(* IEC 61131-3 sources: ae-tiax/test/ParkingCounter, 2 files *)

(* ---- TestCounter.st ---- *)
USING Siemens.Ax.ExampleLibrary;
USING AxUnit;

NAMESPACE Siemens.Ax

    {TestFixture}
    CLASS TestCounter
        VAR
            c : Counter;
            cStateless : Counter;
        END_VAR

        // This method will be called before each test method
        {TestSetup}
        METHOD PUBLIC MyTestSetup
            c := cStateless;
        END_METHOD
        {Test}
        METHOD PUBLIC Test_CountUp_1_Time_And_Get_1
            c.CountUp();
            Assert.Equal(actual := c.GetValue(), expected := 1);
        END_METHOD
        {Test}
        METHOD PUBLIC Test_CountDown_1_Time_And_Get_Minus_1
            c.CountDown();
            Assert.Equal(actual := c.GetValue(), expected := -1);
        END_METHOD
        {Test}
        METHOD PUBLIC Test_CountUp_3_Times_And_Get_3
            c.CountUp();
            c.CountUp();
            c.CountUp();
            Assert.Equal(actual := c.GetValue(), expected := 3);
        END_METHOD
        {Test}
        METHOD PUBLIC Test_CountDown_3_Time_And_Get_Minus_3
            c.CountDown();
            c.CountDown();
            c.CountDown();
            Assert.Equal(actual := c.GetValue(), expected := -3);
        END_METHOD
        {Test}
        METHOD PUBLIC Test_SetValue_To_5_And_Get_5
            c.SetValue(5);
            Assert.Equal(actual := c.GetValue(), expected := 5);
        END_METHOD
        {Test}
        METHOD PUBLIC Test_SetValue_wit_DefaultValue_And_Get_0
            c.SetValue(5);
            c.SetValue();
            Assert.Equal(actual := c.GetValue(), expected := 0);
        END_METHOD
    END_CLASS

END_NAMESPACE

(* ---- TestParkingCounterFB.st ---- *)
USING Siemens.Ax.ExampleLibrary;
USING AxUnit;

NAMESPACE Siemens.Ax

    {TestFixture}
    CLASS TestParkingCounterFB
        VAR
            c : ParkingCounterWrapper;
            cStateless : ParkingCounterWrapper;
            bInside : BOOL;
            bOutside : BOOL;
        END_VAR
        // This method will be called before each test method
        {TestSetup}
        METHOD PUBLIC MyTestSetup
            c := cStateless;
        END_METHOD
        /// Sinal Sequence for 1 object entering
        METHOD Enter_1_object_signal_sequence

            bInside := FALSE;
            bOutside := FALSE;
            c(BSensorOutside := bOutside, BSensorInside := bInside, Limit := 2);
            bInside := FALSE;
            bOutside := TRUE;
            c(BSensorOutside := bOutside, BSensorInside := bInside, Limit := 2);
            bInside := TRUE;
            bOutside := TRUE;
            c(BSensorOutside := bOutside, BSensorInside := bInside, Limit := 2);
            bInside := TRUE;
            bOutside := FALSE;
            c(BSensorOutside := bOutside, BSensorInside := bInside, Limit := 2);
            bInside := FALSE;
            bOutside := FALSE;
            c(BSensorOutside := bOutside, BSensorInside := bInside, Limit := 2);
        END_METHOD
        /// Sinal Sequence for 1 object leaving
        METHOD Leave_1_object_signal_sequence
            bInside := FALSE;
            bOutside := FALSE;
            c(BSensorOutside := bOutside, BSensorInside := bInside, Limit := 2);
            bInside := TRUE;
            bOutside := FALSE;
            c(BSensorOutside := bOutside, BSensorInside := bInside, Limit := 2);
            bInside := TRUE;
            bOutside := TRUE;
            c(BSensorOutside := bOutside, BSensorInside := bInside, Limit := 2);
            bInside := FALSE;
            bOutside := TRUE;
            c(BSensorOutside := bOutside, BSensorInside := bInside, Limit := 2);
            bInside := FALSE;
            bOutside := FALSE;
            c(BSensorOutside := bOutside, BSensorInside := bInside, Limit := 2);
        END_METHOD
        {Test}
        METHOD PUBLIC Count_1_object_entering
            VAR_TEMP
                cv : DINT;
            END_VAR
            THIS.Enter_1_object_signal_sequence();
            cv := c.countValue;
            Assert.Equal(actual := cv, expected := 1);
        END_METHOD
        {Test}
        METHOD PUBLIC CheckLimit_of_to_by_entering_three_objects
            VAR_TEMP
                cv : DINT;
            END_VAR
            THIS.Enter_1_object_signal_sequence();
            THIS.Enter_1_object_signal_sequence();
            THIS.Enter_1_object_signal_sequence();
            cv := c.countValue;
            Assert.Equal(actual := cv, expected := 2);
        END_METHOD
        {Test}
        METHOD PUBLIC Remove_one_of_one_object_and_expect_0
            VAR_TEMP
                cv : DINT;
            END_VAR
            THIS.Enter_1_object_signal_sequence();
            THIS.Leave_1_object_signal_sequence();
            cv := c.countValue;
            Assert.Equal(actual := cv, expected := 0);
        END_METHOD
    END_CLASS

END_NAMESPACE
